FUNCTION_BLOCK fb_Clamp EXTENDS FB_Generic
VAR_INPUT
END_VAR
VAR_OUTPUT
END_VAR
VAR
	iClampDn1: INT;

	iClampUp1: INT;
	iClampUp2: INT;
	fbClampHeight	:AIN_EL3004;
	flag00: BOOL;
	flag01: BOOL;
	fbClampLock	:FB_ClampLock;
	fbClampUnlock	:FB_ClampUnlock;
	M_ClampUnlock: INT;
	fbClampJog	:FB_ClampJog;
	httss: REAL;
	test1	:INT;
	test2	:INT;
	height	:REAL;
	tmpMid,tmpFrnt,tmpRear	:BOOL;
	
	rtClampLock0: r_trig;
	i1,i2,i3,i4	:INT;
	
	fbClampMove	:FB_ClampMove;
	aa: INT;
	rtExLight: R_trig;
	ftExLight: f_trig;
	rtClampMove: R_trig;
	rtExTopSlide: R_trig;
	rtExBtmSlide: R_trig;
END_VAR

SUPER^();

//fbClampHeight(Enable:=TRUE , In:=ANALOG_in_ClampHeight , MaxOut:=CNST_CLAMP_MAXCONVERT ,Offset:=0,  OutData=> );
//ANALOG_in_ClampHeight	:=test1;
stFolder.ClampPress	:=40.0*TO_REAL(ANALOG_in_PumpPress)/32767;
stFolder.ClampHt_ActPos	:=Anolog_To_Height(value:= ANALOG_in_ClampHeight);
stFolder.Status.Clamp_AtPressPoint	:= stFolder.ClampPress > CNST_CLAMP_LIGHT_PRESSURE_SETPOINT;
stFolder.Status.Clamp_LtHalfPoint	:= stFolder.ClampHt_ActPos <= stFolderPara.ClampHalfPos;
stFolder.Status.Clamp_AtZeroPoint	:= stFolder.ClampHt_ActPos < CONST_CLAMP_POS_CALIBRATION;
stFolder.Status.Clamp_GtLowPoint	:= stFolder.ClampHt_ActPos > stFolderPara.Clamp_LowPos;

flag00:=stFolder.Status.Slitter_AtHome AND stFolder.Status.ApronTopFold_AtHome AND stFolder.Status.ApronBtmFold_AtHome;
flag01:=flag00 AND (stFolder.Status.Table_AtHome OR stFolder.Status.Flip_AtWork) AND (stFolder.Status.Feed_AtHome OR (stFolder.Status.Feed_AtWork AND stFolder.ClampHt_ActPos > 60 ));
fbClampLock(Rst:=rtReset.Q);
fbClampUnlock(Rst:=rtReset.Q);

httss	:=Anolog_To_Height(value:=test1 );
test2	:=Height_To_Anology(height:= height);

(*-----------------------------------------------------------------------------------*)
(*------------------------- Clamp Gauge Front/Rear/Middle ---------------------------*)
(*-----------------------------------------------------------------------------------*)
rtExLight(CLK:=Hmi_bArray[1] , Q=> );
ftExLight(CLK:=Hmi_bArray[1] , Q=> );
rtExTopSlide(CLK:=stFolder.Status.ApronTopSlide_AtWork , Q=> );
rtExBtmSlide(CLK:=stFolder.Status.ApronBtmSlide_AtWork , Q=> );
IF rtExLight.Q THEN
	fbClampMove.Ex	:=TRUE;
	fbClampMove._iHeavyGauge	:=0;
END_IF
IF ftExLight.Q OR (NOT Hmi_bArray[1] AND (rtExTopSlide.Q OR rtExBtmSlide.Q)) THEN
	fbClampMove.Ex	:=TRUE;
	IF stFolder.Status.ApronTopSlide_AtWork AND NOT stFolder.Status.ApronBtmSlide_AtWork THEN
		fbClampMove._iHeavyGauge	:=+1;
	ELSIF stFolder.Status.ApronBtmSlide_AtWork AND NOT stFolder.Status.ApronTopSlide_AtWork THEN
		fbClampMove._iHeavyGauge	:=-1;
	END_IF
END_IF

IF NOT Hmi_bArray[1] AND (fbUnitModeManager.eModeStatus=ePMLUnitMode_SemiAuto OR fbUnitModeManager.eModeStatus=ePMLUnitMode_Auto ) THEN
	fbClampMove._iHeavyGauge	:=stFolderCom.paraClampMove;
	fbClampMove.Ex	:=stFolderCom.TaskClamp=eTask_ClampMove;
END_IF
		
		
fbClampMove(Ex:= , UnitMode:= , Done=> );
rtClampMove(CLK:=fbClampMove.Done , Q=> );
IF rtClampMove.Q THEN
	stFolderCom.TaskClamp :=eTask_NULL;
END_IF

ACTION A_AutoRun:

END_ACTION

ACTION A_ManualRun:
fbClampJog(Rst:=rtReset.Q);
END_ACTION

ACTION A_SemiAuto:
rtClampLock0(CLK:=fbClampLock.Done , Q=> );

IF stFolderCom.TaskClamp =eTask_ClampLock AND flag01 THEN
	fbClampLock.Ex		:=TRUE;
	fbClampLock.para	:=stFolderCom.paraClamp;
	IF rtClampLock0.Q THEN 
		stFolderCom.TaskClamp	:=eTask_NULL;
		fbClampLock.Ex		:=FALSE;
	END_IF;
	
ELSIF stFolderCom.TaskClamp = eTask_ClampUnlock AND flag00 THEN
	fbClampUnLock.Ex	:=TRUE;
	fbClampUnlock.para	:=stFolderCom.paraClamp;
	IF fbClampUnlock.Done THEN
		stFolderCom.TaskClamp	:=eTask_NULL;
		fbClampUnLock.Ex	:=FALSE;
	END_IF
ELSIF stFolderCom.TaskClamp = eTask_ClampJog THEN
	fbClampJog(Rst:=rtReset.Q);
ELSIF stFolderCom.TaskClamp =eTask_NULL THEN
	fbClampLock.Ex		:=FALSE;
	fbClampUnLock.Ex	:=FALSE;
END_IF
END_ACTION

{attribute 'object_name' := 'M_Execute'}
METHOD M_Execute
CASE fbUnitModeManager.eModeStatus OF
	ePMLProtUnitMode_Production:		//Production
		;
	ePMLProtUnitMode_Maintenance:		
		//
		;
		ePMLUnitMode_Auto:
		A_SemiAuto();
	ePMLUnitMode_SemiAuto:
		A_SemiAuto();
	ePMLUnitMode_AutoSlitter:
		A_SemiAuto();
	ePMLProtUnitMode_Manual:		//Manual
		A_ManualRun();
		
		
		

		
END_CASE
END_METHOD

END_FUNCTION_BLOCK

(* stored: Version 1.1.0.1, ProductVersion 3.1.4024.15
   POU fb_Clamp: Id {cf1c3620-cfb7-4ba2-8c92-21d36f17440d}, SpecialFunc None
   Action A_AutoRun: Id {25268d4f-1f4a-4138-a01c-46224cda0929}
   Action A_ManualRun: Id {044d2078-e6a7-4883-8ac4-ba2bc572e5e4}
   Action A_SemiAuto: Id {8f5b2cdf-cbae-48ed-9f58-bb181c24af9a}
   Method M_Execute: Id {3dce9d6d-6211-4703-b00b-4bef74d92804} *)
